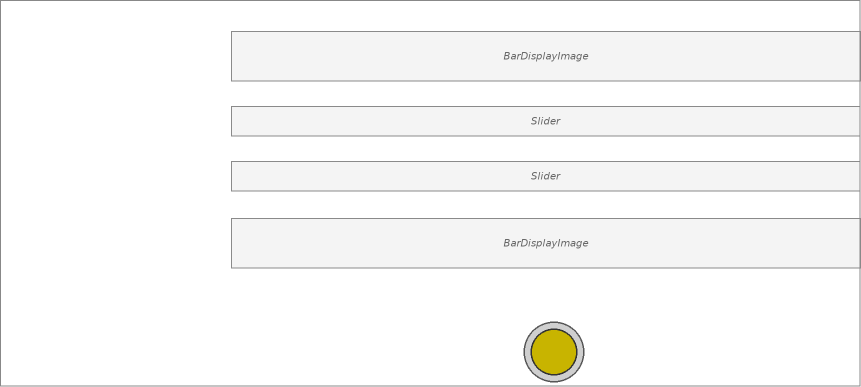
VISUALIZATION Visu  // 861x387
    Slider (231,106 629x30), variable: MAIN.nPot1, scale 10..30
    Slider (231,161 629x30), variable: MAIN.nPot2, scale -30..40
    Lamp1 (519,317 70x70), variable: MAIN.bL1, style: Lamp-Lamp1-Yellow
    BarDisplayImage (231,31 630x50), value: MAIN.nPot1, style: BarDisplayImage-Gray, scale format: %.1f, scale 10..30
    BarDisplayImage (231,218 630x50), value: MAIN.nPot2, style: BarDisplayImage-Gray, scale format: %.1f, scale -30..40
END_VISUALIZATION

(* stored: Version 1.1.0.1, ProductVersion 3.1.4024.12
   Visu Visu: Id {3827c7be-3a31-47dc-b96f-5cf0597dbac9} *)
